FUNCTION_BLOCK FB_CONTROL
VAR_INPUT
	Start:BOOL;
END_VAR
VAR_OUTPUT
	McOutputs:ST_McOutputs;
END_VAR
VAR
	MoveAbsolute:MC_MoveAbsolute;
END_VAR

VAR_IN_OUT
	Axis: AXIS_REF;
END_VAR

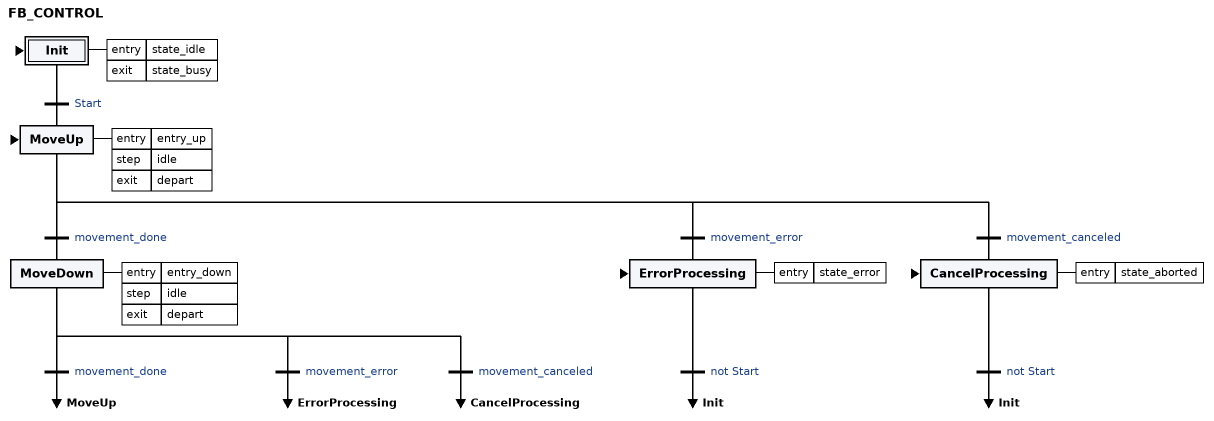
INITIAL_STEP Init:
    state_idle(P1);  // entry action
    state_busy(P0);  // exit action
END_STEP
TRANSITION FROM Init TO MoveUp
    := Start;
END_TRANSITION
STEP MoveUp:
    entry_up(P1);  // entry action
    idle(N);  // step action
    depart(P0);  // exit action
END_STEP
TRANSITION FROM MoveUp TO MoveDown
    := movement_done;
END_TRANSITION
TRANSITION FROM MoveUp TO ErrorProcessing
    := movement_error;
END_TRANSITION
STEP ErrorProcessing:
    state_error(P1);  // entry action
END_STEP
TRANSITION FROM ErrorProcessing TO Init
    := not Start;
END_TRANSITION
TRANSITION FROM MoveUp TO CancelProcessing
    := movement_canceled;
END_TRANSITION
STEP CancelProcessing:
    state_aborted(P1);  // entry action
END_STEP
TRANSITION FROM CancelProcessing TO Init
    := not Start;
END_TRANSITION
STEP MoveDown:
    entry_down(P1);  // entry action
    idle(N);  // step action
    depart(P0);  // exit action
END_STEP
TRANSITION FROM MoveDown TO MoveUp
    := movement_done;
END_TRANSITION
TRANSITION FROM MoveDown TO ErrorProcessing
    := movement_error;
END_TRANSITION
TRANSITION FROM MoveDown TO CancelProcessing
    := movement_canceled;
END_TRANSITION

ACTION depart:
MoveAbsolute.Execute:=FALSE;
idle();
END_ACTION

ACTION entry_down:
MoveAbsolute.Position:=0;
MoveAbsolute.Velocity:=100;
MoveAbsolute.Execute:=TRUE;
END_ACTION

ACTION entry_up:
MoveAbsolute.Position:=1000;
MoveAbsolute.Velocity:=100;
MoveAbsolute.Execute:=TRUE;
END_ACTION

ACTION idle:
MoveAbsolute(
	Axis:= Axis, 
	Execute:= , 
	Position:= , 
	Velocity:= , 
	Acceleration:= , 
	Deceleration:= , 
	Jerk:= , 
	BufferMode:= MC_Aborting, 
	Options:= , 
	Done=> , 
	Busy=> , 
	Active=> , 
	CommandAborted=> , 
	Error=> , 
	ErrorID=> );
END_ACTION

TRANSITION movement_canceled:
MoveAbsolute.CommandAborted;
END_TRANSITION

TRANSITION movement_done:
MoveAbsolute.Done;
END_TRANSITION

TRANSITION movement_error:
MoveAbsolute.Error;
END_TRANSITION

ACTION state_aborted:
McOutputs.CommandAborted:=TRUE;
McOutputs.Done:=
McOutputs.Busy:=
McOutputs.Active:=
McOutputs.Error:=FALSE;
McOutputs.ErrorID:=0;
END_ACTION

ACTION state_busy:
McOutputs.Busy:=TRUE;
McOutputs.Active:=
McOutputs.CommandAborted:=
McOutputs.Done:=
McOutputs.Error:=FALSE;
McOutputs.ErrorID:=0;
END_ACTION

ACTION state_done:
McOutputs.Busy:=
McOutputs.Active:=
McOutputs.CommandAborted:=
McOutputs.Done:=
McOutputs.Error:=FALSE;
McOutputs.ErrorID:=0;
END_ACTION

ACTION state_error:
McOutputs.Busy:=
McOutputs.Active:=
McOutputs.CommandAborted:=
McOutputs.Done:=FALSE;
McOutputs.Error:=TRUE;
McOutputs.ErrorID:=MoveAbsolute.ErrorID;
END_ACTION

ACTION state_idle:
McOutputs.Done:=TRUE;
McOutputs.Busy:=
McOutputs.Active:=
McOutputs.CommandAborted:=
McOutputs.Error:=FALSE;
McOutputs.ErrorID:=0;
END_ACTION

END_FUNCTION_BLOCK

(* stored: Version 1.1.0.1, ProductVersion 3.1.4024.9
   POU FB_CONTROL: Id {284f8d3f-5f13-4896-b59e-2754bc062bab}, SpecialFunc None
   Action depart: Id {b009ea50-3abb-4302-878f-b9c2d10aa9bf}
   Action entry_down: Id {5eca5aa6-ac68-4244-89f4-3410067c089f}
   Action entry_up: Id {08b1b4a5-8a2b-4068-a18f-0e3ec348ae37}
   Action idle: Id {75d38ec5-6e17-43d2-85a1-cac53520a068}
   Transition movement_canceled: Id {7a002748-3ade-4db3-94ba-ff0bba6110e7}
   Transition movement_done: Id {227d8fb7-8301-4b58-b09d-8afb8258a018}
   Transition movement_error: Id {550af31a-f5bd-4a25-a34c-69818a3c9f1f}
   Action state_aborted: Id {509c218a-1f02-42fd-8d6f-6ada493cfdfc}
   Action state_busy: Id {eff2e806-2560-45b4-a209-14fc32475238}
   Action state_done: Id {3bb3f80f-abf9-4f5e-ba95-8b09a67caa16}
   Action state_error: Id {6ab1f0e1-e7a8-4a07-982d-7aeb463425a5}
   Action state_idle: Id {ca06cae6-fd77-4edb-b3ed-50f7c9bb0fce} *)
